Fanuc KAREL source: kf00043.KL

-- PROVISIONAL review KL for V770-1; original PC SHA256 46ca7bca6a9219790379df4ba865bd1facaf646e508cb38e7d20fc915ba094e1
-- Incomplete behavior may be omitted. Consult companion uncertainty JSON. Do not deploy.
PROGRAM KF00043
%NOLOCKGROUP
VAR
  I : INTEGER
  J : INTEGER
  X : REAL
  Y : REAL
  B : BOOLEAN
  C : BOOLEAN
  TXT : STRING[80]
  TXT2 : STRING[80]
  STATUS : INTEGER
-- UNRESOLVED_DECL AI type=002010
-- UNRESOLVED_DECL BI type=002010
-- UNRESOLVED_DECL P type=000102
-- UNRESOLVED_DECL JP type=000199
-- UNRESOLVED_DECL PF type=000101
-- UNRESOLVED_DECL V1 type=000013
-- UNRESOLVED_DECL V2 type=000013
-- UNRESOLVED_DECL REC type=001100
BEGIN
  -- UNRESOLVED_PC offsets 5-20; opcodes 2E,22,32,35
  -- UNRESOLVED_PC offsets 25-41; opcodes 22,32,34,23
  -- UNRESOLVED_PC offsets 46-50; opcodes 7F
END KF00043
